FUNCTION_BLOCK PCA_TRANSF
  {SET_ATTRIBUTE(OpcUa, SERVICE)}
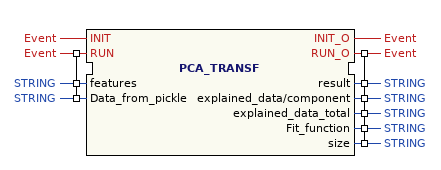
  EVENT_INPUT
    INIT;
    RUN WITH features, Data_from_pickle; {SET_ATTRIBUTE(OpcUa, Method)}
  END_EVENT
  EVENT_OUTPUT
    INIT_O;
    RUN_O WITH result, explained_data/component, explained_data_total, Fit_function, size;
  END_EVENT
  VAR_INPUT
    features : STRING; {SET_ATTRIBUTE(OpcUa, Variable.RUN)}
    Data_from_pickle : STRING; {SET_ATTRIBUTE(OpcUa, Variable.RUN)}
  END_VAR
  VAR_OUTPUT
    result : STRING; {SET_ATTRIBUTE(OpcUa, Variable.RUN)}
    explained_data/component : STRING; {SET_ATTRIBUTE(OpcUa, Variable.RUN)}
    explained_data_total : STRING; {SET_ATTRIBUTE(OpcUa, Variable.RUN)}
    Fit_function : STRING; {SET_ATTRIBUTE(OpcUa, Variable.RUN)}
    size : STRING; {SET_ATTRIBUTE(OpcUa, Variable.RUN)}
  END_VAR
END_FUNCTION_BLOCK
